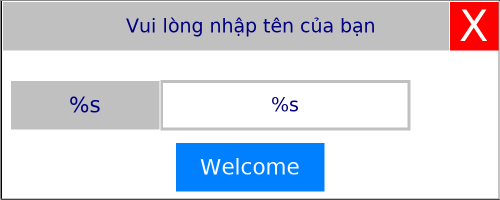
VISUALIZATION startpage  // 500x200
    Rectangle (1,0 500x200)
    Rectangle (2,1 498x50), "Vui lòng nhập tên của bạn"
    Rectangle (160,80 250x50), "%s", text variable: username
        OnMouseDown: write username via VisuDialogs.Keypad
    Rectangle (175,142 150x50), "Welcome", invisible if: not openstartpage, input disabled if: not openstartpage
        OnMouseDown: CloseDialog Dialog=startpage, Result=OK, NumpadKeypadSet=True
        OnMouseDown: change screen: N_Setting_Line1
    Rectangle (449,1 50x50), "X"
        OnMouseDown: CloseDialog Dialog=startpage, Result=OK, NumpadKeypadSet=True
    Rectangle (10,80 150x50), "%s", text variable: getuser
END_VISUALIZATION

(* stored: Version 1.1.0.1, ProductVersion 3.1.4024.12
   Visu startpage: Id {94976436-1fa0-497b-9436-db4b48524220} *)
